{attribute addProperty BoxType "EL1918-0000-0016"}
{attribute addProperty Id "FSoE_InputsFSoE_Inputs_4B31FBCB567FSoE_OutputsFSoE_Outputs_6E970715486"}
{attribute addProperty CRC "3822512082"}
{attribute addProperty SizeInBites "104"}
{attribute addProperty SizeInBytes "13"}
TYPE Module_1_FSOE_E3D6E7D2 :
STRUCT
	{attribute addProperty Name "FSoE_Inputs"}
	FSoE_Inputs  : FSoE_Inputs_4B31FBCB;
	{attribute addProperty Name "FSoE_Outputs"}
	FSoE_Outputs  : FSoE_Outputs_6E970715;
END_STRUCT
END_TYPE

(* stored: Version 1.2.0.0, ProductVersion 3.1.4024.9
   DUT Module_1_FSOE_E3D6E7D2: Id {91294b38-0586-49ab-bbf6-44a35952515a} *)
